(* PLC project Unnamed, Unknown Unnamed 1 *)
(* stored: creationDateTime 2025-06-21T17:41:03, modificationDateTime 2025-06-21T18:08:38 *)

PROGRAM sr_rs
  VAR
    input1 AT %IX100.0 : BOOL;
    input2 AT %IX100.1 : BOOL;
    reset AT %IX100.2 : BOOL;
    load AT %IX100.3 : BOOL;
    output1 AT %QX100.0 : BOOL;
    output2 AT %QX100.1 : BOOL;
  END_VAR
  VAR
    RS0 : RS;
    SR0 : SR;
  END_VAR

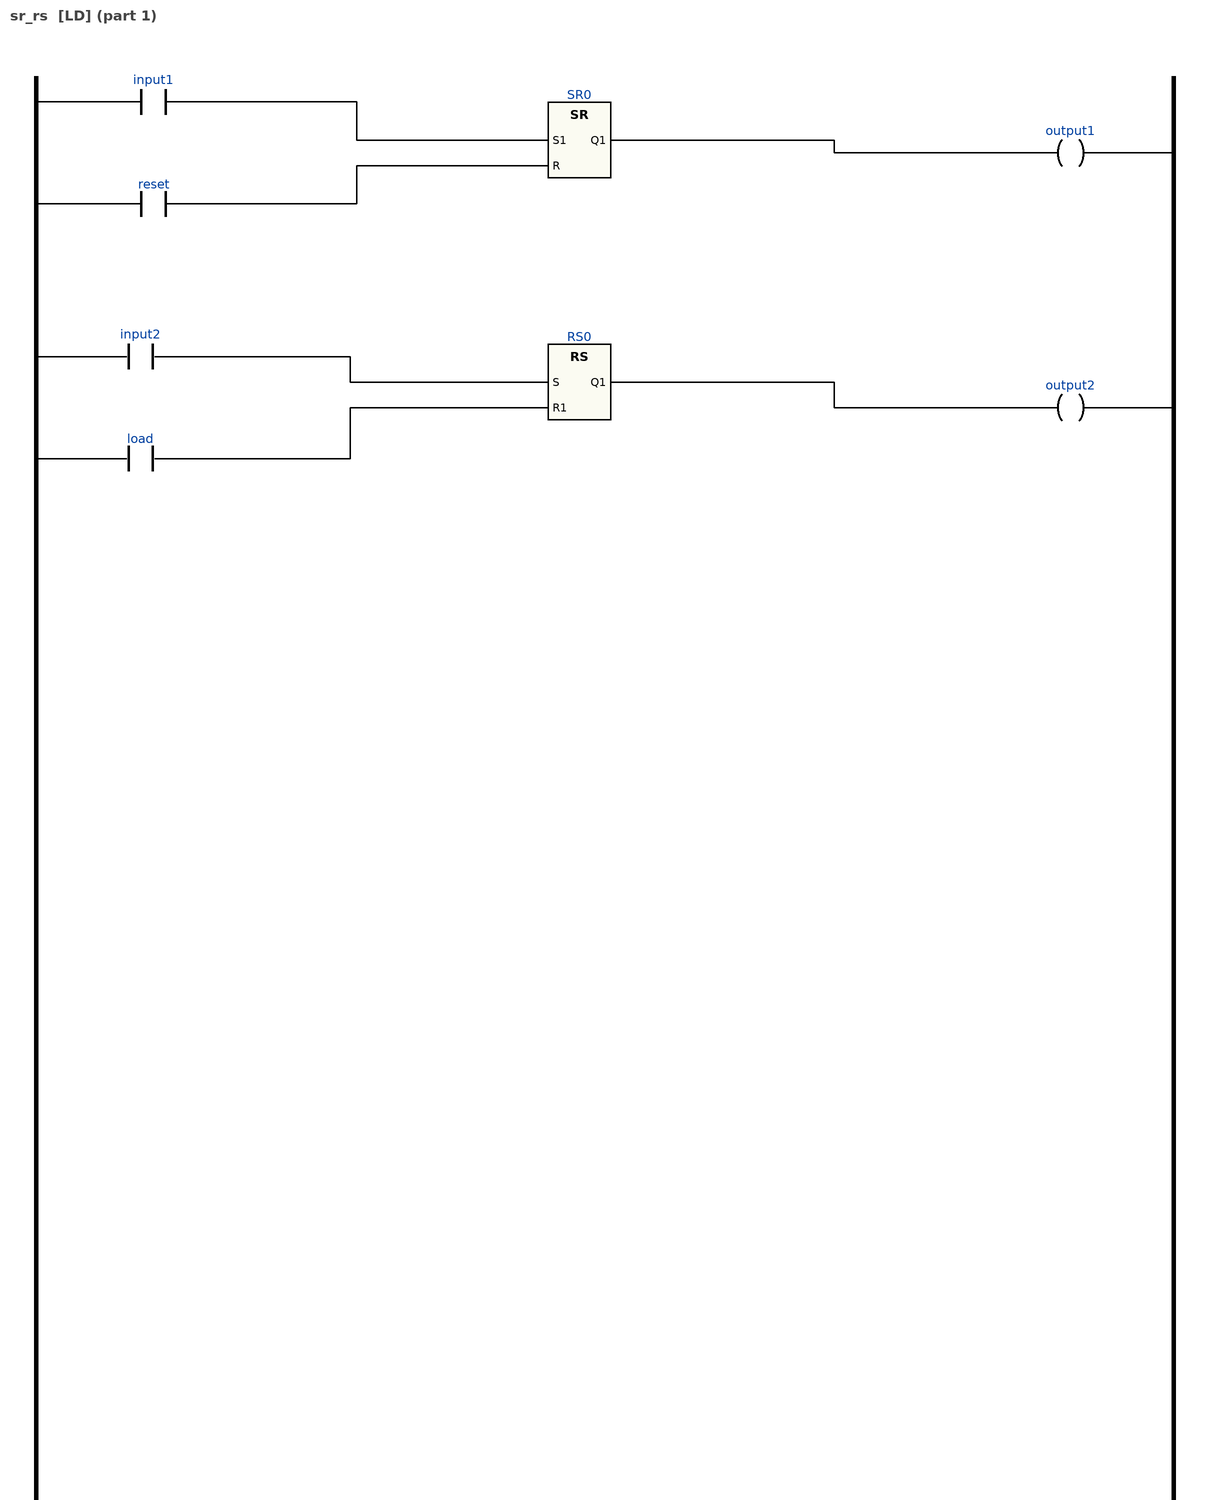
(* LD diagram, written out as Structured Text *)
SR0(S1 := input1, R := reset);
output1 := SR0.Q1;
RS0(S := input2, R1 := load);
output2 := RS0.Q1;
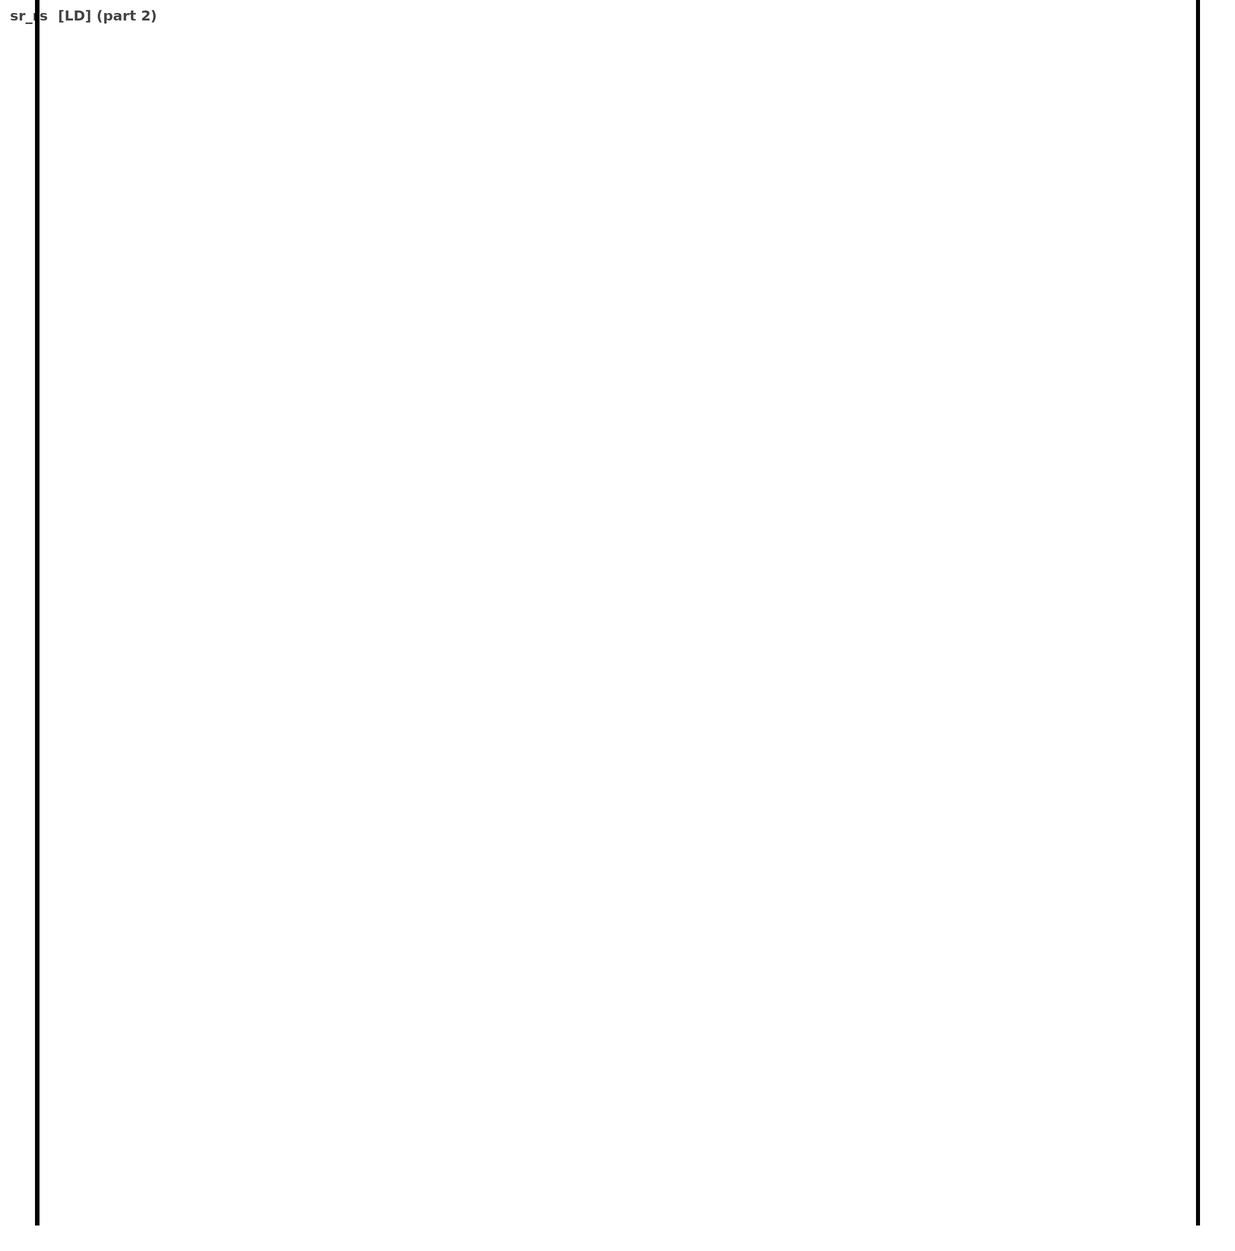
END_PROGRAM

CONFIGURATION Config0
  RESOURCE Res0 ON PLC
    TASK task0(INTERVAL := T#20ms, PRIORITY := 0);
    PROGRAM instance0 WITH task0 : sr_rs;
  END_RESOURCE
END_CONFIGURATION
